{attribute 'no_explicit_call' := 'do not call this POU directly'}
//{attribute 'hide_all_locals'}
// Function Block to invoke RPC calls.
FUNCTION_BLOCK FINAL FB_RPC IMPLEMENTS I_RpcArguments, I_RpcInvoke, I_RpcReleaseHandle

VAR
	sAmsNetId 			: T_AmsNetId := GCL.cLocalAmsNetId;
	nAmsPort			: T_AmsPort;
	nSymbolHandle 		: UDINT;
	sSymbol				: T_MaxString;
END_VAR

VAR
	fbRdWrReq 				: ADSRDWRT;
	fbAdsWrReqRelHandle 	: ADSWRITE; 
	nHandleToRelease		: UDINT := cNoSymbolNameHandle;	
	eStep				: ( HNDBYNAME, VALBYHND, RELEASEHND) := HNDBYNAME;
	eArgs				: ( NO_LOCK, LOCK ) := NO_LOCK;
	fbArguments			: FB_ArgumentsBuffer;
	tAdsTMOUT			: TIME := GCL.cAdsTimeOut;
END_VAR

VAR CONSTANT
	cNoSymbolNameHandle : UDINT := 0;
END_VAR

METHOD Argument : I_RpcArguments
VAR_INPUT
	anyArg	: ANY;
END_VAR
VAR
	stAny : ST_AnyType;
	eAdsErr : E_AdsErr;
END_VAR
Argument := THIS^;

IF eArgs = LOCK THEN
	RETURN;
END_IF

stAny.pValue := anyArg.pValue;
stAny.nSize := anyArg.diSize;

eAdsErr := fbArguments.SetArgument(stAny);
IF eAdsErr <> E_AdsErr.NOERR THEN
	RETURN;
END_IF
END_METHOD

METHOD FB_exit : BOOL
VAR_INPUT
	bInCopyCode : BOOL; // if TRUE, the exit method is called for exiting an instance that is copied afterwards (online change).
END_VAR
IF nSymbolHandle > cNoSymbolNameHandle THEN
	ReleaseHandle();
END_IF
END_METHOD

METHOD FB_init : BOOL
VAR_INPUT
    bInitRetains 	: BOOL; // if TRUE, the retain variables are initialized (warm start / cold start)
    bInCopyCode  	: BOOL; // if TRUE, the instance afterwards gets moved into the copy code (online change)
	sAmsNetId		: T_AmsNetID;
	nAmsPort		: T_AmsPort;
	sInstancePath	: STRING;	// e.g. MAIN.fbYourFB
	sSymbol			: STRING;	// e.g. YourSymbolName
END_VAR
Initialize();

IF bInCopyCode THEN
	ReleaseHandle();
END_IF


IF sAmsNetId = '' THEN
	THIS^.sAmsNetId := GCL.cLocalAmsNetId;
ELSE
	THIS^.sAmsNetId := sAmsNetId;
END_IF

THIS^.nAmsPort := nAmsPort;
THIS^.sSymbol := sSymbol;

THIS^.sSymbol := F_RpcSymbol(sInstancePath, sSymbol);
END_METHOD

METHOD PRIVATE GetSymbolHandleByName : ST_AdsStatus
VAR_INPUT
	sNetId 		: REFERENCE TO T_AmsNetId;
	nPort		: T_AmsPort;
	sSymbol		: REFERENCE TO T_MaxString;
END_VAR
fbRdWrReq(
	NETID:= sNetId, 
	PORT:= nPort, 
	IDXGRP:= ADSIGRP_SYM_HNDBYNAME, 
	IDXOFFS:= 16#0, 
	WRITELEN:= TO_UDINT(LEN(sSymbol)), 
	READLEN:= SIZEOF(nSymbolHandle), 
	SRCADDR:= ADR(sSymbol), 
	DESTADDR:= ADR(nSymbolHandle), 
	WRTRD:= TRUE, 
	TMOUT:= tAdsTMOUT, 
	BUSY=> GetSymbolHandleByName.bBusy, 
	ERR=> GetSymbolHandleByName.bError, 
	ERRID=> GetSymbolHandleByName.nError);
END_METHOD

METHOD PRIVATE Initialize
VAR_INPUT
END_VAR
ResetArguments();
nHandleToRelease := cNoSymbolNameHandle;
fbAdsWrReqRelHandle(WRITE:= FALSE);
fbRdWrReq(WRTRD:= FALSE);
eArgs := NO_LOCK;
END_METHOD

METHOD Invoke : ST_AdsStatus

VAR
	stRetVal : ST_AdsStatus;
END_VAR
eArgs := LOCK;

CASE eStep OF
	HNDBYNAME:
		Invoke.bBusy := TRUE;
		stRetVal := GetSymbolHandleByName(sAmsNetId, nAmsPort, sSymbol);
		IF NOT stRetVal.bBusy AND NOT stRetVal.bError THEN
			fbRdWrReq(WRTRD:= FALSE);
			eStep:= VALBYHND;
		ELSE
			Invoke := stRetVal;
			eStep := HNDBYNAME;
			RETURN;
		END_IF
		
	VALBYHND:
		Invoke := ReadValueByHandle(fbArguments.pArgsBuffer,
									fbArguments.nArgsLength, 
									fbArguments.pRetValBuffer, 
									fbArguments.nRetValLength);		
		IF NOT Invoke.bBusy THEN
			eArgs := NO_LOCK;
			IF NOT Invoke.bError THEN
				Invoke.nError := fbArguments.GetRetVal();
				Invoke.bError := Invoke.nError <> E_AdsErr.NOERR;
			END_IF;
			fbRdWrReq(WRTRD:= FALSE);
			ResetArguments();
			IF Invoke.bError AND Invoke.nError = E_AdsErr.DEVICE_NOTIFYHNDINVALID THEN
				Invoke.bBusy := TRUE;
				Invoke.bError := FALSE;
				Invoke.nError := E_AdsErr.NOERR;
				eStep := HNDBYNAME;
			END_IF
		END_IF
END_CASE;
END_METHOD

METHOD NoReturnValue : I_RpcInvoke
NoReturnValue := THIS^;
END_METHOD

METHOD PRIVATE ReadValueByHandle : ST_AdsStatus
VAR_INPUT
	pArgs		: PVOID;
	nLenArgs 	: UDINT;
	pRetVal		: PVOID;
	nLenRetVal 	: UDINT;
END_VAR

VAR
	nNullDummy 	: UDINT;
END_VAR

IF pArgs = NULL THEN
	pArgs := ADR(nNullDummy);
	nLenArgs := 0;
END_IF
	
IF pRetVal = NULL THEN
	pRetVal := ADR(nNullDummy);
	nLenRetVal := 0;
END_IF

fbRdWrReq(
		IDXGRP:= ADSIGRP_SYM_VALBYHND, 
		IDXOFFS:= nSymbolHandle, 
		WRITELEN:=nLenArgs, 
		READLEN:= nLenRetVal , 
		SRCADDR:= pArgs, 
		DESTADDR:= pRetVal, 
		WRTRD:= TRUE, 
		TMOUT:= tAdsTMOUT, 
		BUSY=> ReadValueByHandle.bBusy, 
		ERR=> ReadValueByHandle.bError, 
		ERRID=> ReadValueByHandle.nError);
END_METHOD

METHOD ReleaseHandle : ST_AdsStatus
IF THIS^.nSymbolHandle = cNoSymbolNameHandle THEN
	RETURN;
END_IF

IF nHandleToRelease = cNoSymbolNameHandle THEN
	fbAdsWrReqRelHandle(WRITE:= FALSE);
	nHandleToRelease := THIS^.nSymbolHandle;
END_IF

fbAdsWrReqRelHandle(
	NETID:= THIS^.sAmsNetId, 
	PORT:= THIS^.nAmsPort, 
	IDXGRP:= ADSIGRP_SYM_RELEASEHND, 
	IDXOFFS:= 16#0, 
	LEN:= SIZEOF(nHandleToRelease), 
	SRCADDR:= ADR(nHandleToRelease), 
	WRITE:= TRUE, 
	TMOUT:= tAdsTMOUT, 
	BUSY=> ReleaseHandle.bBusy, 
	ERR=> ReleaseHandle.bError, 
	ERRID=> ReleaseHandle.nError);
	
IF NOT fbAdsWrReqRelHandle.BUSY OR fbAdsWrReqRelHandle.ERR THEN
	eStep := HNDBYNAME;
	nHandleToRelease := cNoSymbolNameHandle;	
END_IF
END_METHOD

METHOD PRIVATE ResetArguments
VAR_INPUT
END_VAR
fbArguments.Reset();
END_METHOD

METHOD ReturnValue : I_RpcInvoke
VAR_INPUT
	anyRetVal	: ANY;
END_VAR
VAR
	stAny : ST_AnyType;
END_VAR
ReturnValue := THIS^;

IF eArgs = LOCK THEN
	RETURN;
END_IF

IF anyRetVal.diSize <= 0 THEN
	RETURN;
END_IF

stAny.pValue := anyRetVal.pValue;
stAny.nSize := anyRetVal.diSize;

fbArguments.SetRetVal(stAny);
END_METHOD

PROPERTY tAdsTimeOut : TIME
GET
tAdsTimeOut := tAdsTMOUT;
END_GET
SET
IF tAdsTimeout > T#0MS THEN
	tAdsTMOUT := tAdsTimeOut;
END_IF
END_SET
END_PROPERTY

METHOD VarInOut : I_RpcArguments
VAR_INPUT
	anyArg	: ANY;
END_VAR

VAR
	stAny : ST_AnyType;
	eAdsErr : E_AdsErr;
END_VAR
VarInOut := THIS^;

IF eArgs = LOCK THEN
	RETURN;
END_IF

IF anyArg.diSize <= 0 THEN
	RETURN;
END_IF

stAny.pValue := anyArg.pValue;
stAny.nSize := anyArg.diSize;

eAdsErr := fbArguments.SetVarInOut(stAny);
IF eAdsErr <> E_AdsErr.NOERR THEN
	RETURN;
END_IF
END_METHOD

END_FUNCTION_BLOCK

(* stored: Version 1.1.0.1, ProductVersion 3.1.4024.12
   POU FB_RPC: Id {4ee15778-936c-4cfb-8f05-eb32519906ab}, SpecialFunc None
   Folder ITFs: Id {668e42c6-659c-4814-8136-a732fd2d063a}
   Method Argument: Id {17a0b69b-5e8e-462a-9d38-6c479fb154bc}
   Method FB_exit: Id {623ea868-fbdc-450e-bc05-7c3f6fe62930}
   Method FB_init: Id {c158b92d-f079-4fd5-bc01-d1513e1d0acf}
   Method GetSymbolHandleByName: Id {c9e2504e-3556-4f2c-af7a-893a12908fd2}
   Method Initialize: Id {c87535b2-cb59-4680-8a4e-d44d93bf7cf8}
   Method Invoke: Id {8851f7d7-adbe-4317-9571-95d25ada74e0}
   Method NoReturnValue: Id {8bd51905-f529-4121-a95b-bf2c0e80eb14}
   Method ReadValueByHandle: Id {4ce6f1ab-ddd9-485f-a2ba-6f0da58cd7d5}
   Method ReleaseHandle: Id {744fe4e4-969e-4cb9-ad4d-b05680ad0542}
   Method ResetArguments: Id {91d66985-f93c-4427-bdfe-fa7879f2ade4}
   Method ReturnValue: Id {9077a3e1-4e93-49ea-8e46-4e884568ccfb}
   Property tAdsTimeOut: Id {ab711797-88bd-4976-ab5a-b05750afb586}
   Get Get: Id {d1c33412-a6dc-4123-a09c-a3c20614ed14}
   Set Set: Id {a73f1060-b87e-4fca-9592-045718ff207c}
   Method VarInOut: Id {838ed4a6-f966-4780-9212-1601030fa5d6} *)
